// TIA Portal project "IntermittenzaDoppioTimer" (V18)

(* hardware
DEVICE "Stazione S7-1500/ET200MP_1"  S7-1500 station
   slot 0: "Telaio di montaggio_0"  Rack  6ES7 590-1***0-0AA0
   slot 1: "PLC_1"  CPU 1511-1 PN  6ES7 511-1AL03-0AB0  V3.0
      slot 3: "Display CPU_1"  6ES7591-1AA00-0AA0
      slot 32768: "Interfaccia PROFINET_1"  X1
         slot 32769: "Porta_1"  X1 P1
         slot 32770: "Porta_2"  X1 P2
      slot 34817: "Virtual CP interface port_1"  Virtual CP interface port  Virtual CP interface port
*)

// ===== PLC "PLC_1"  CPU 1511-1 PN =====

VAR_GLOBAL   // PLC tag table "Tabella delle variabili standard"
   "Attiva_Pos1" AT %M0.0 : Bool;
   "Intermittenza_Attivata" AT %M0.1 : Bool;
   "Comando-Pos1" AT %M0.3 : Bool;
   "Comando-Pos2" AT %M0.4 : Bool;
   "Attiva_Pos2" AT %M0.7 : Bool;
   "timePos1_ON" AT %MD8 : Time;
   "timePos2_ON" AT %MD12 : Time;
END_VAR

// folder: System blocks/Program resources

DATA_BLOCK "Pos2_Timer_ON"   // DB2
{ S7_Optimized_Access := 'TRUE' }
AUTHOR : Simatic
FAMILY : IEC
NAME : IEC_TMR
VERSION : 1.0
// stored: InstanceOfName IEC_TIMER
"IEC_TIMER"
BEGIN
END_DATA_BLOCK

DATA_BLOCK "Pos1_Timer_ON"   // DB4
{ S7_Optimized_Access := 'TRUE' }
AUTHOR : Simatic
FAMILY : IEC
NAME : IEC_TMR
VERSION : 1.0
// stored: InstanceOfName IEC_TIMER
"IEC_TIMER"
BEGIN
END_DATA_BLOCK

// folder: (top level)

ORGANIZATION_BLOCK "Main"   // OB1, LAD, ProgramCycle
TITLE = "Main Program Sweep (Cycle)"
{ S7_Optimized_Access := 'TRUE' }
VERSION : 0.1
   VAR_INPUT
      Initial_Call : Bool;   // Initial call of this OB
      Remanence : Bool;   // =True, if remanent data are available
   END_VAR
BEGIN

REGION Network 1: Comando Attiva/Disattiva Intermittenza
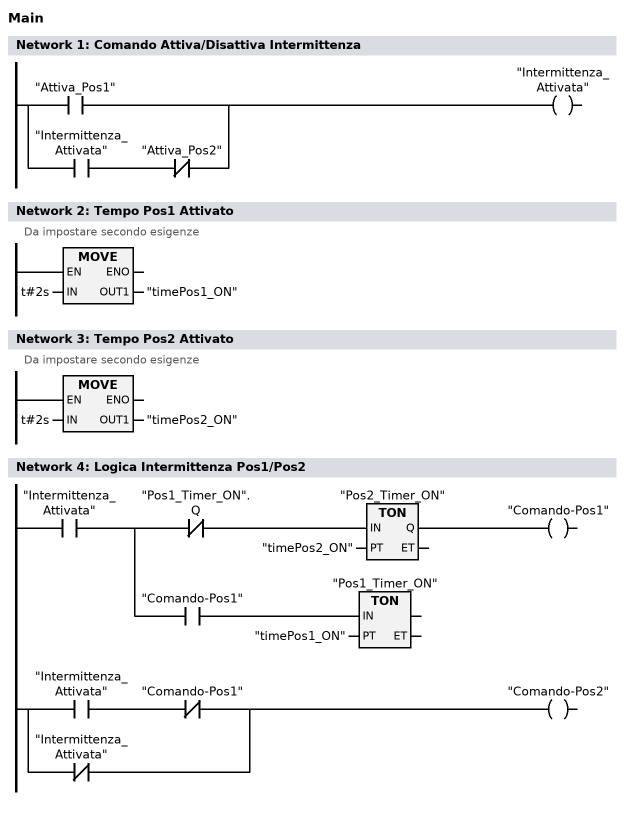
   RUNG wire#powerrail
      Contact( "Attiva_Pos1" )
      wire#w1
      Coil( "Intermittenza_Attivata" )
   END_RUNG
   RUNG wire#powerrail
      Contact( "Intermittenza_Attivata" )
      I_Contact( "Attiva_Pos2" )
   END_RUNG wire#w1
   // the same network as SCL:
   "Intermittenza_Attivata" := "Attiva_Pos1" OR ("Intermittenza_Attivata" AND NOT "Attiva_Pos2");
END_REGION

REGION Network 2: Tempo Pos1 Attivato
   // Da impostare secondo esigenze
   RUNG wire#powerrail
      Move(in := t#2s, out1 => "timePos1_ON")
   END_RUNG
   // the same network as SCL:
   "timePos1_ON" := t#2s;
END_REGION

REGION Network 3: Tempo Pos2 Attivato
   // Da impostare secondo esigenze
   RUNG wire#powerrail
      Move(in := t#2s, out1 => "timePos2_ON")
   END_RUNG
   // the same network as SCL:
   "timePos2_ON" := t#2s;
END_REGION

REGION Network 4: Logica Intermittenza Pos1/Pos2
   "Pos2_Timer_ON".TON(IN := "Intermittenza_Attivata" AND NOT "Pos1_Timer_ON".Q, PT := "timePos2_ON");
   "Comando-Pos1" := "Pos2_Timer_ON".Q;
   "Pos1_Timer_ON".TON(IN := "Intermittenza_Attivata" AND "Comando-Pos1", PT := "timePos1_ON");
   "Comando-Pos2" := ("Intermittenza_Attivata" AND NOT "Comando-Pos1") OR NOT "Intermittenza_Attivata";
END_REGION
END_ORGANIZATION_BLOCK